FUNCTION CONCAT4 : T_MaxString
VAR_INPUT
	STR1	:T_MaxString;
	STR2	:T_MaxString;
	STR3	:T_MaxString;
	STR4	:T_MaxString;
END_VAR
VAR
	_MainString	:T_MaxString:='';
END_VAR

_MainString:=CONCAT(STR1:=STR1,STR2:=STR2);
_MainString:=CONCAT(STR1:=_MainString,STR2:=STR3);
_MainString:=CONCAT(STR1:=_MainString,STR2:=STR4);

CONCAT4:=_MainString;

END_FUNCTION

(* stored: Version 1.1.0.1, ProductVersion 3.1.4024.6
   POU CONCAT4: Id {82e3861f-d1b5-480f-82db-58859773693d}, SpecialFunc None *)
